(* IEC 61131-3 sources: Industry-PLC-LLM/data/PLCBEAD_repo/PLCBEAD_PLCEmbed-main/PLC-BEAD/Source/GEB/MANUAL, 1 file *)

(* ---- MANUAL.ST ---- *)
FUNCTION MANUAL:BOOL

	VAR_INPUT
		_IN :	BOOL;
		_ON :	BOOL;
		OFF :	BOOL;
	END_VAR

	MANUAL := NOT OFF AND (_IN OR _ON);

END_FUNCTION

PROGRAM program0
	VAR
		_IN :	BOOL;
		_ON :	BOOL;
		OFF :	BOOL;

		OUT : BOOL;
	END_VAR

	OUT := MANUAL(_IN, _ON, OFF);

END_PROGRAM
